Staubli VAL3: start.pgx

program start()
begin
  call createTask()
  userPage()
  cls()
  put("Hello World!")
  gotoxy(0,1)
  put("Opening Connection...")
end
